{attribute 'GeneratedUsingTerminal: EJ1914-0000-0017'}
{attribute addProperty BoxType "EJ1914-0000-0017"}
{attribute addProperty Id "FSoE_InputsFSoE_Inputs_8952FEF011FSoE_OutputsFSoE_Outputs_7E6724397"}
{attribute addProperty CRC "1427501450"}
{attribute addProperty Size "18"}
TYPE Module_1_FSOE_5515F18A :
STRUCT
	{attribute addProperty Name "FSoE_Inputs"}
	FSoE_Inputs  : FSoE_Inputs_8952FEF0;
	{attribute addProperty Name "FSoE_Outputs"}
	FSoE_Outputs  : FSoE_Outputs_7E672439;
END_STRUCT
END_TYPE

(* stored: Version 1.2.0.0, ProductVersion 3.1.4024.9
   DUT Module_1_FSOE_5515F18A: Id {e4de2049-99c0-464c-96fe-5ad948a3dcf6} *)
